{attribute 'qualified_only'}
{attribute 'strict'}
{attribute 'to_string'}
TYPE E_BaseEvents_Category :
(
	None		:= 0,
	Error		:= 1, 
	Alarm		:= 2, 
	Safety		:= 3, 
	Message		:= 4

);
END_TYPE

(* stored: Version 1.1.0.1
   DUT E_BaseEvents_Category: Id {aee22ca8-38f0-4d5e-8215-120a4a034c27} *)
